// TIA Portal V18 export
// export: Created 2026-03-12T16:04:35.0623994Z, ExportSetting WithDefaults, DisplayName Totally Integrated Automation Portal, DisplayVersion V18 Update 5, DisplayName TIA Portal Openness, DisplayVersion V18 Update 5, DisplayName TIA Portal Version Control Interface, DisplayVersion V18, DisplayName SINAMICS Startdrive Advanced, DisplayVersion V18, DisplayName SINAMICS Startdrive G130, G150, S120, S150, SINAMICS MV, S210, DisplayVersion V18, DisplayName SINAMICS Startdrive G110M, G120, G120C, G120D, G120P, G115D, DisplayVersion V18, DisplayName STEP 7 Professional, DisplayVersion V18 Update 5, DisplayName STEP 7 Safety, DisplayVersion V18, DisplayName WinCC Professional, DisplayVersion V18 Update 5
FUNCTION_BLOCK "FB CONDIÇÃO DE PARTIDA"   // FB6, LAD
TITLE = Function Block CONDIÇÃO DE PARTIDA - Intertravamentos para partir o motor/bomba
{ S7_Optimized_Access := 'TRUE' }
VERSION : 0.1
// Network 1: Gerenciamento Status Motor/Bomba
// Network 2: Recebimento dos sinais de entrada (Sinais de campo e comandos)
// Network 3: MODO MANUAL: Conjunto de condições para ligar e desligar
// Network 4: MODO AUTOMÁTICO: Conjunto de condições para ligar e desligar
// Network 5: FALHA: Condicionamento de falha
// Network 6: LIGA BOMBA: Validando intertravamentos para ligar
// stored: AutoNumber true, IsIECCheckEnabled false, IsRetainMemResEnabled false, MemoryReserve 100, SetENOAutomatically false, UDAEnableTagReadback false
   VAR_INPUT
      INPUT_LIGADO : Bool;   // 1 = Sinal elétrico de campo indicando bomba ligada
      INPUT_DESLIGADO : Bool;   // 1 = Sinal elétrico de campo indicando bomba desligada
      INPUT_FALHA : Bool;   // 0 = Sinal elétrico de campo indicando bomba em falha
      INPUT_LOCAL : Bool;   // 1 = Sinal elétrico de campo indicando bomba em local
      INPUT_REMOTO : Bool;   // 1 = Sinal elétrico de campo indicando bomba em remoto
      INPUT_LOC_AUTO : Bool;   // 1 = Sinal elétrico de campo indicando bomba em local automático
      INPUT_FALHA_PROFINET : Bool;   // 1 = Indica falta de comunicação PROFINET com o equipamento
      INPUT_HABILITA_LIGA_AUTO : Bool;   // 1 = Sinal para habilitar Liga Bomba em Modo Automático quando todas as condições foram atentidas
      CMD_LIGA : Bool;   // Comando enviado da IHM/SCADA para ligar a bomba
      CMD_MANUTEN : Bool;   // Comando enviado da IHM/SCADA para colocar a bomba em Modo de Manutenção
      CMD_MODO : Bool;   // Comando enviado da IHM/SCADA para colocar a bomba em (0 = Modo Manual, 1 = Modo Automático)
   END_VAR
   VAR_OUTPUT
      STATUS_MOTOR : Byte;   // 0 = DESLIGADO; 1 = LIGADO; 2 = FALHA; 3 = MANUTENÇÃO; 4 = SEM COMUNICAÇÃO MODBUS
      LIGA_BOMBA : Bool;   // Saída acionada para ligar a bomba remotamente
      REMOTO_MAN : Bool;   // Saída para indicar bomba em Remoto Manual
      REMOTO_AUTO : Bool;   // Saída para indicar bomba em Remoto Automático
      LOCAL_MAN : Bool;   // Saída para indicar bomba em Local Manual
   END_VAR
   VAR
      MANUTEN : Bool;   // Variável local para Indicar bomba em Modo Manutenção
      REMOTO : Bool;   // Variável local para indicar bomba em Modo Remoto
      FALHA : Bool;   // Variável local para indicar bomba em Falha
      LOCAL_AUTO : Bool;   // Variável local para indicar bomba em Modo Local Automático
      LIGA_REM_MAN : Bool;   // Variável local para Acionamento Remoto Manual
      LIGA_REM_AUTO : Bool;   // Variável local para Acionamento Remoto Automático
   END_VAR
   VAR_TEMP   // added for the SCL form of the ladder/FBD networks
      _w1 : Bool;
   END_VAR
BEGIN

REGION Network 1: Recebimento dos sinais de entrada (Sinais de campo e comandos)
   // INPUT_ABERTA = Entrada de sinal de Bomba Ligada
   // INPUT_FECHADA = Entrada de sinal de Bomba Desligada
   // INPUT_FALHA = Entrada de sinal de Bomba em Falha
   // INPUT_FALHA_PROFINET = Sem comunicação Profinet
   // STATUS_MOTOR: 0 = DESLIGADO; 1 = LIGADO; 2 = FALHA; 3 = MANUTENÇÃO; 4 = SEM COMUNICAÇÃO MODBUS
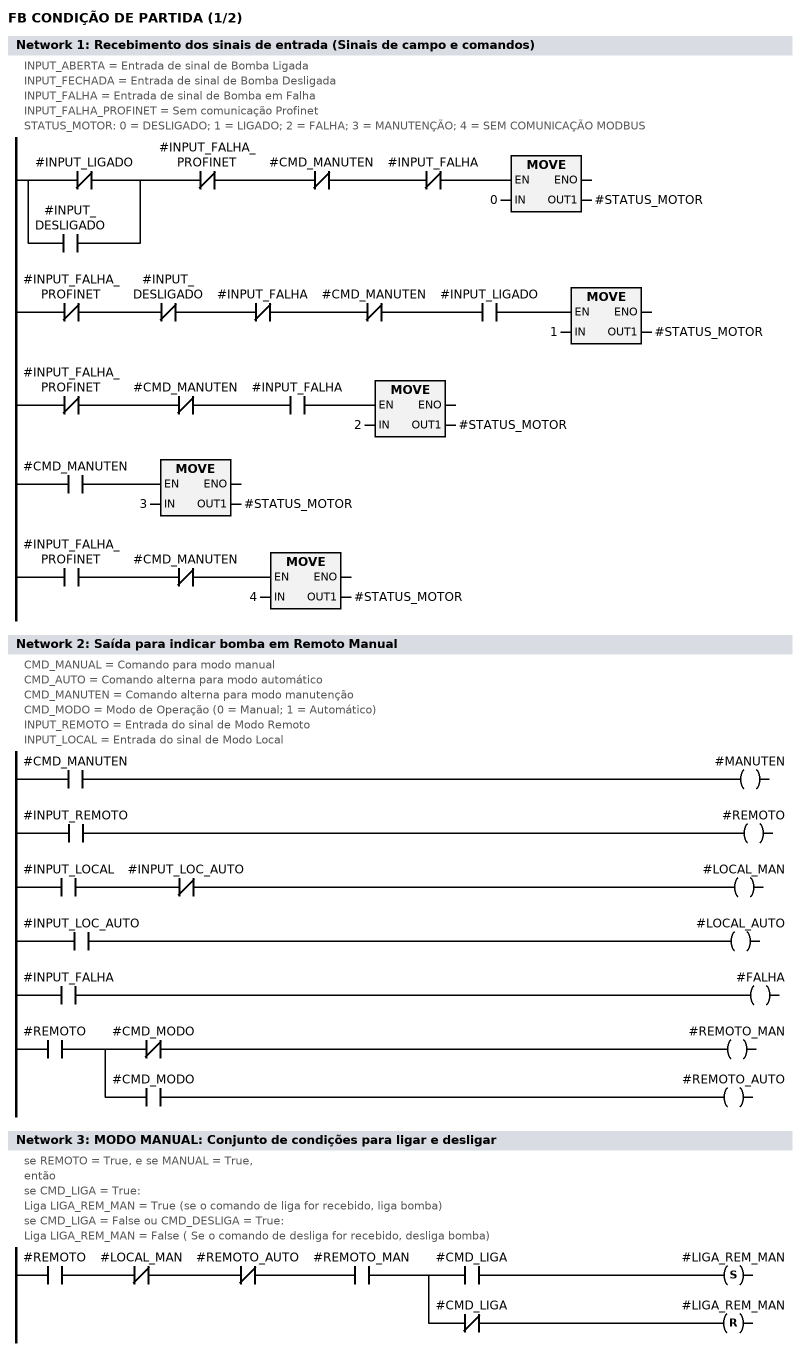
   RUNG wire#powerrail
      I_Contact( #INPUT_LIGADO )
      wire#w1
      I_Contact( #INPUT_FALHA_PROFINET )
      I_Contact( #CMD_MANUTEN )
      I_Contact( #INPUT_FALHA )
      Move(in := 0, out1 => #STATUS_MOTOR)
   END_RUNG
   RUNG wire#powerrail
      Contact( #INPUT_DESLIGADO )
   END_RUNG wire#w1
   RUNG wire#powerrail
      I_Contact( #INPUT_FALHA_PROFINET )
      I_Contact( #INPUT_DESLIGADO )
      I_Contact( #INPUT_FALHA )
      I_Contact( #CMD_MANUTEN )
      Contact( #INPUT_LIGADO )
      Move(in := 1, out1 => #STATUS_MOTOR)
   END_RUNG
   RUNG wire#powerrail
      I_Contact( #INPUT_FALHA_PROFINET )
      I_Contact( #CMD_MANUTEN )
      Contact( #INPUT_FALHA )
      Move(in := 2, out1 => #STATUS_MOTOR)
   END_RUNG
   RUNG wire#powerrail
      Contact( #CMD_MANUTEN )
      Move(in := 3, out1 => #STATUS_MOTOR)
   END_RUNG
   RUNG wire#powerrail
      Contact( #INPUT_FALHA_PROFINET )
      I_Contact( #CMD_MANUTEN )
      Move(in := 4, out1 => #STATUS_MOTOR)
   END_RUNG
   // the same network as SCL:
   IF (NOT #INPUT_LIGADO OR #INPUT_DESLIGADO) AND NOT #INPUT_FALHA_PROFINET AND NOT #CMD_MANUTEN AND NOT #INPUT_FALHA THEN
       #STATUS_MOTOR := 0;
   END_IF;
   IF NOT #INPUT_FALHA_PROFINET AND NOT #INPUT_DESLIGADO AND NOT #INPUT_FALHA AND NOT #CMD_MANUTEN AND #INPUT_LIGADO THEN
       #STATUS_MOTOR := 1;
   END_IF;
   IF NOT #INPUT_FALHA_PROFINET AND NOT #CMD_MANUTEN AND #INPUT_FALHA THEN #STATUS_MOTOR := 2; END_IF;
   IF #CMD_MANUTEN THEN #STATUS_MOTOR := 3; END_IF;
   IF #INPUT_FALHA_PROFINET AND NOT #CMD_MANUTEN THEN #STATUS_MOTOR := 4; END_IF;
END_REGION

REGION Network 2: Saída para indicar bomba em Remoto Manual
   // CMD_MANUAL = Comando para modo manual
   // CMD_AUTO = Comando alterna para modo automático
   // CMD_MANUTEN = Comando alterna para modo manutenção
   // CMD_MODO = Modo de Operação (0 = Manual; 1 = Automático)
   // INPUT_REMOTO = Entrada do sinal de Modo Remoto
   // INPUT_LOCAL = Entrada do sinal de Modo Local
   RUNG wire#powerrail
      Contact( #CMD_MANUTEN )
      Coil( #MANUTEN )
   END_RUNG
   RUNG wire#powerrail
      Contact( #INPUT_REMOTO )
      Coil( #REMOTO )
   END_RUNG
   RUNG wire#powerrail
      Contact( #INPUT_LOCAL )
      I_Contact( #INPUT_LOC_AUTO )
      Coil( #LOCAL_MAN )
   END_RUNG
   RUNG wire#powerrail
      Contact( #INPUT_LOC_AUTO )
      Coil( #LOCAL_AUTO )
   END_RUNG
   RUNG wire#powerrail
      Contact( #INPUT_FALHA )
      Coil( #FALHA )
   END_RUNG
   RUNG wire#powerrail
      Contact( #REMOTO )
      wire#w1
      I_Contact( #CMD_MODO )
      Coil( #REMOTO_MAN )
   END_RUNG
   RUNG wire#w1
      Contact( #CMD_MODO )
      Coil( #REMOTO_AUTO )
   END_RUNG
   // the same network as SCL:
   #MANUTEN := #CMD_MANUTEN;
   #REMOTO := #INPUT_REMOTO;
   #LOCAL_MAN := #INPUT_LOCAL AND NOT #INPUT_LOC_AUTO;
   #LOCAL_AUTO := #INPUT_LOC_AUTO;
   #FALHA := #INPUT_FALHA;
   #REMOTO_MAN := #REMOTO AND NOT #CMD_MODO;
   #REMOTO_AUTO := #REMOTO AND #CMD_MODO;
END_REGION

REGION Network 3: MODO MANUAL: Conjunto de condições para ligar e desligar
   // se REMOTO = True, e se MANUAL = True,
   // 
   // então
   // se CMD_LIGA = True: 
   // Liga LIGA_REM_MAN = True (se o comando de liga for recebido, liga bomba)
   // 
   // se CMD_LIGA = False ou CMD_DESLIGA = True:
   // Liga LIGA_REM_MAN = False ( Se o comando de desliga for recebido, desliga bomba)
   RUNG wire#powerrail
      Contact( #REMOTO )
      I_Contact( #LOCAL_MAN )
      I_Contact( #REMOTO_AUTO )
      Contact( #REMOTO_MAN )
      wire#w1
      Contact( #CMD_LIGA )
      S_Coil( #LIGA_REM_MAN )
   END_RUNG
   RUNG wire#w1
      I_Contact( #CMD_LIGA )
      R_Coil( #LIGA_REM_MAN )
   END_RUNG
   // the same network as SCL:
   #_w1 := #REMOTO AND NOT #LOCAL_MAN AND NOT #REMOTO_AUTO AND #REMOTO_MAN;
   IF #_w1 AND #CMD_LIGA THEN #LIGA_REM_MAN := TRUE; END_IF;
   IF #_w1 AND NOT #CMD_LIGA THEN #LIGA_REM_MAN := FALSE; END_IF;
END_REGION

REGION Network 4: Variável local para Acionamento Remoto Auto
   // se REMOTO = True, e se AUTO = True:
   // 
   // então
   // se LIGA_REM_AUTO = True:
   // e se PARAMETRO < PARAMETRO_LIGA;
   // então LIGA_REM_AUTO = True (se a leitura for menor que o cadastro para ligar, liga em remoto automático)
   // 
   // se LIGA_REM_AUTO = False:
   // e se PARAMETRO >= PARAMETRO_DESLIGA:
   // então Desliga REMOTO AUTOMÁTICO (se a leitura for maior ou igual ao cadastro para desligar, desliga em remoto automático)
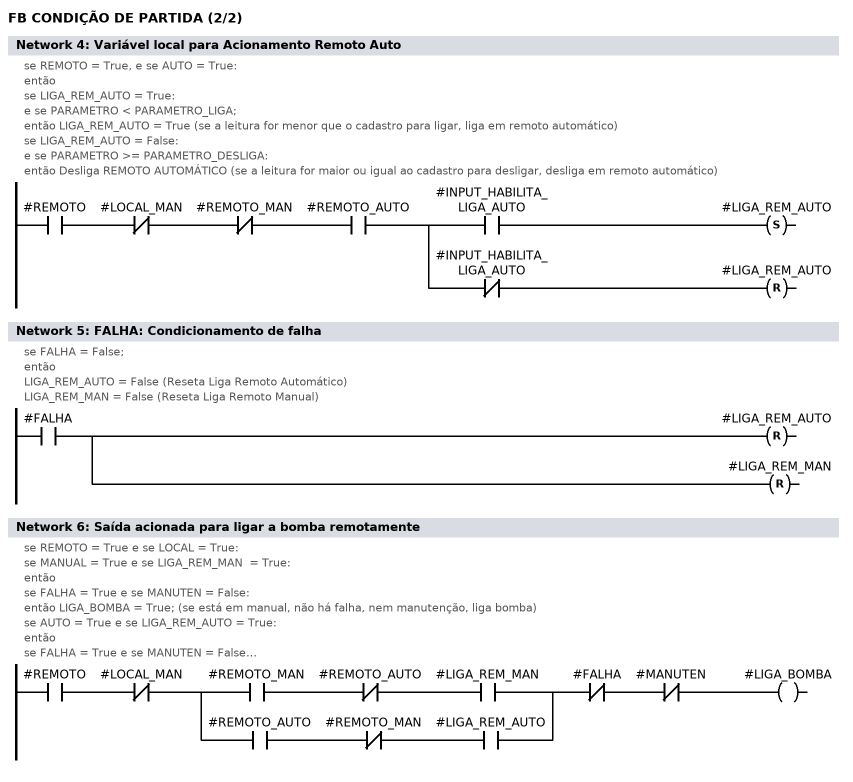
   RUNG wire#powerrail
      Contact( #REMOTO )
      I_Contact( #LOCAL_MAN )
      I_Contact( #REMOTO_MAN )
      Contact( #REMOTO_AUTO )
      wire#w1
      Contact( #INPUT_HABILITA_LIGA_AUTO )
      S_Coil( #LIGA_REM_AUTO )
   END_RUNG
   RUNG wire#w1
      I_Contact( #INPUT_HABILITA_LIGA_AUTO )
      R_Coil( #LIGA_REM_AUTO )
   END_RUNG
   // the same network as SCL:
   #_w1 := #REMOTO AND NOT #LOCAL_MAN AND NOT #REMOTO_MAN AND #REMOTO_AUTO;
   IF #_w1 AND #INPUT_HABILITA_LIGA_AUTO THEN #LIGA_REM_AUTO := TRUE; END_IF;
   IF #_w1 AND NOT #INPUT_HABILITA_LIGA_AUTO THEN #LIGA_REM_AUTO := FALSE; END_IF;
END_REGION

REGION Network 5: FALHA: Condicionamento de falha
   // se FALHA = False;
   // 
   // então
   // LIGA_REM_AUTO = False (Reseta Liga Remoto Automático)
   // LIGA_REM_MAN = False (Reseta Liga Remoto Manual)
   RUNG wire#powerrail
      Contact( #FALHA )
      wire#w1
      R_Coil( #LIGA_REM_AUTO )
   END_RUNG
   RUNG wire#w1
      R_Coil( #LIGA_REM_MAN )
   END_RUNG
   // the same network as SCL:
   IF #FALHA THEN
       #LIGA_REM_AUTO := FALSE;
       #LIGA_REM_MAN := FALSE;
   END_IF;
END_REGION

REGION Network 6: Saída acionada para ligar a bomba remotamente
   // se REMOTO = True e se LOCAL = True:
   // 
   // se MANUAL = True e se LIGA_REM_MAN  = True:
   // então
   // se FALHA = True e se MANUTEN = False:
   // então LIGA_BOMBA = True; (se está em manual, não há falha, nem manutenção, liga bomba)
   // 
   // se AUTO = True e se LIGA_REM_AUTO = True:
   // então
   // se FALHA = True e se MANUTEN = False:
   // então LIGA_BOMBA = True; (se está em automático, não há falha, nem manutenção, liga bomba)
   RUNG wire#powerrail
      Contact( #REMOTO )
      I_Contact( #LOCAL_MAN )
      wire#w1
      Contact( #REMOTO_MAN )
      I_Contact( #REMOTO_AUTO )
      Contact( #LIGA_REM_MAN )
      wire#w2
      I_Contact( #FALHA )
      I_Contact( #MANUTEN )
      Coil( #LIGA_BOMBA )
   END_RUNG
   RUNG wire#w1
      Contact( #REMOTO_AUTO )
      I_Contact( #REMOTO_MAN )
      Contact( #LIGA_REM_AUTO )
   END_RUNG wire#w2
   // the same network as SCL:
   #LIGA_BOMBA := #REMOTO AND NOT #LOCAL_MAN AND ((#REMOTO_MAN AND NOT #REMOTO_AUTO AND #LIGA_REM_MAN) OR (#REMOTO_AUTO AND NOT #REMOTO_MAN AND #LIGA_REM_AUTO)) AND NOT #FALHA AND NOT #MANUTEN;
END_REGION
END_FUNCTION_BLOCK
